// LS Electric XG5000 project: 동남120
// PLC NewPLC
// module base 0 slot 0: 입출력 모듈:XBC-DN/DP14E (DC 24V 입력 8점, 트랜지스터 출력 6점)

PROGRAM NewProgram (task: 스캔 프로그램)

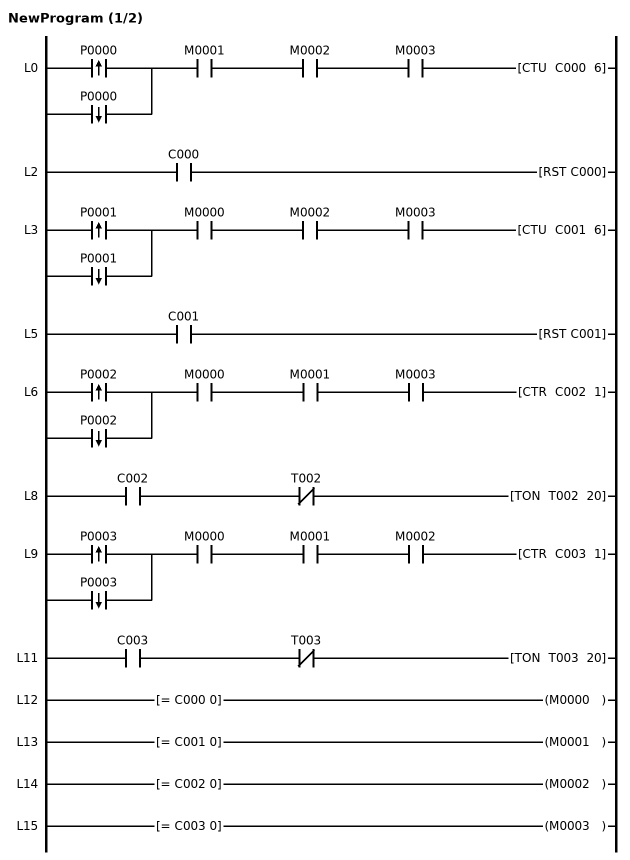
; L0
LOADP     P0000
ORN       P0000
AND       M0001
AND       M0002
AND       M0003
CTU       C000 6
; L2
LOAD      C000
RST       C000
; L3
LOADP     P0001
ORN       P0001
AND       M0000
AND       M0002
AND       M0003
CTU       C001 6
; L5
LOAD      C001
RST       C001
; L6
LOADP     P0002
ORN       P0002
AND       M0000
AND       M0001
AND       M0003
CTR       C002 1
; L8
LOAD      C002
AND NOT   T002
TON       T002 20
; L9
LOADP     P0003
ORN       P0003
AND       M0000
AND       M0001
AND       M0002
CTR       C003 1
; L11
LOAD      C003
AND NOT   T003
TON       T003 20
; L12
LOAD=     C000 0
OUT       M0000
; L13
LOAD=     C001 0
OUT       M0001
; L14
LOAD=     C002 0
OUT       M0002
; L15
LOAD=     C003 0
OUT       M0003

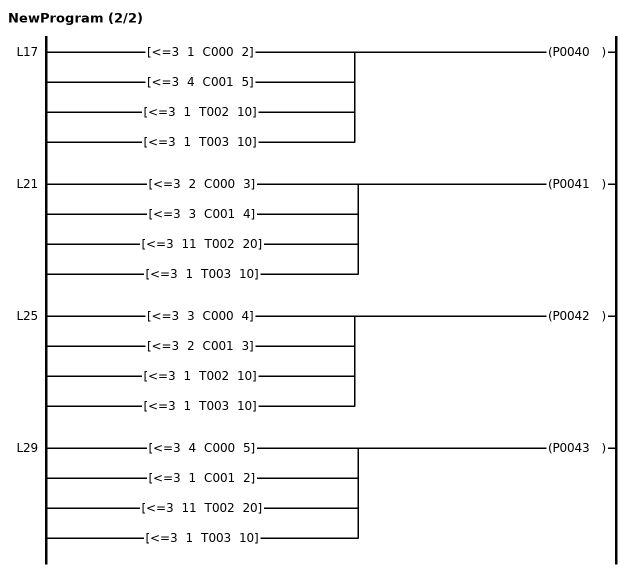
; L17
LOAD<=3   1 C000 2
OR<=3     4 C001 5
OR<=3     1 T002 10
OR<=3     1 T003 10
OUT       P0040
; L21
LOAD<=3   2 C000 3
OR<=3     3 C001 4
OR<=3     11 T002 20
OR<=3     1 T003 10
OUT       P0041
; L25
LOAD<=3   3 C000 4
OR<=3     2 C001 3
OR<=3     1 T002 10
OR<=3     1 T003 10
OUT       P0042
; L29
LOAD<=3   4 C000 5
OR<=3     1 C001 2
OR<=3     11 T002 20
OR<=3     1 T003 10
OUT       P0043